{attribute 'qualified_only'}
{attribute 'strict'}
{attribute 'to_string'}
TYPE LOAD_STATE :
(
	NOT_LOADED,
	LOADING,
	LOADED,
	FAILED
);
END_TYPE

(* stored: Version 1.1.0.1
   DUT LOAD_STATE: Id {85b749e0-aa94-4cb5-999a-d1d66e19b5cf} *)
